FUNCTION_BLOCK FB_Bloque
VAR_INPUT
	Tcheck: TIME := T#1S;
	Treset: TIME := T#1S;
	Tdesplazador: TIME := T#1S;
	Tcinta: TIME := T#0.5S;
END_VAR
VAR_OUTPUT
END_VAR
VAR
	Ciclos: INT;
	Aceptados:INT;
	Rechazados: INT;
	Restantes: INT;
	
	pieza_ok: BOOL;
	
	//Terminal 2
	Pulsador_parada_emergencia AT %I*: BOOL;
	Selector_modo_manual AT %I*: BOOL;
	Pulsador_marcha AT %I*: BOOL;
	Pulsador_parada_NC AT %I*: BOOL;
	Parte_operativa_conectada AT %I*: BOOL;
	Presencia_pale AT %I*: BOOL;
	Codigo_pale_bit_0 AT %I*: BOOL;
	Codigo_pale_bit_1 AT %I*: BOOL;
	
	
	//Terminal 3
	Codigo_pale_bit_2 AT %I*: BOOL;
	Detector_presion AT %I*: BOOL;
	
	//Terminal 4
	Desconecta_parte_operativa AT %Q*: BOOL;
	Lampara_alarma AT %Q*: BOOL;
	Lampara_marcha AT %Q*: BOOL;
	Lampara_falta_material AT %Q*: BOOL;
	Activa_marcha_motor_cinta AT %Q*: BOOL;
	Invierte_marcha_motor_cinta AT %Q*: BOOL;
	Retenedor_pale_baja AT %Q*: BOOL;
	Separador_pale_sube AT %Q*: BOOL;
	
	
	//Terminal 5
 	Avisador_sonoro AT %Q*: BOOL;
	
	//Terminal 6
	Horizontal_descargador_detras AT %I*: BOOL;
	Horizontal_descargador_delante AT %I*: BOOL;
	Vertical_descargador_arriba AT %I*: BOOL;
	Vertical_descargador_abajo AT %I*: BOOL;
	Verificador_arriba AT %I*: BOOL;
	Verificador_abajo AT %I*: BOOL;
	Desplazador_detras AT %I*: BOOL;
	Alimentador_detras AT %I*: BOOL;
	
	
	//Terminal 7
	Alimentador_delante AT %I*: BOOL;
	Vacio_obtenido_vacuostato_descargador AT %I*: BOOL;
	Base_en_Alimentador AT %I*: BOOL;
	
	//Terminal 8
	Descargador_adelante AT %Q*: BOOL;
	Descargador_atras AT %Q*: BOOL;
	Descargador_baja AT %Q*: BOOL;
	Rechazador_adelante AT %Q*: BOOL;
	Verificador_baja AT %Q*: BOOL;
	Desplazador_adelante AT %Q*: BOOL;
	Alimentador_adelante AT %Q*: BOOL;
	Eyector_succiona AT %Q*: BOOL;
	
	NOLAMP: INT;
	t: INT;
	NOTSOUND: INT;
	NOTFOUND: INT;
END_VAR

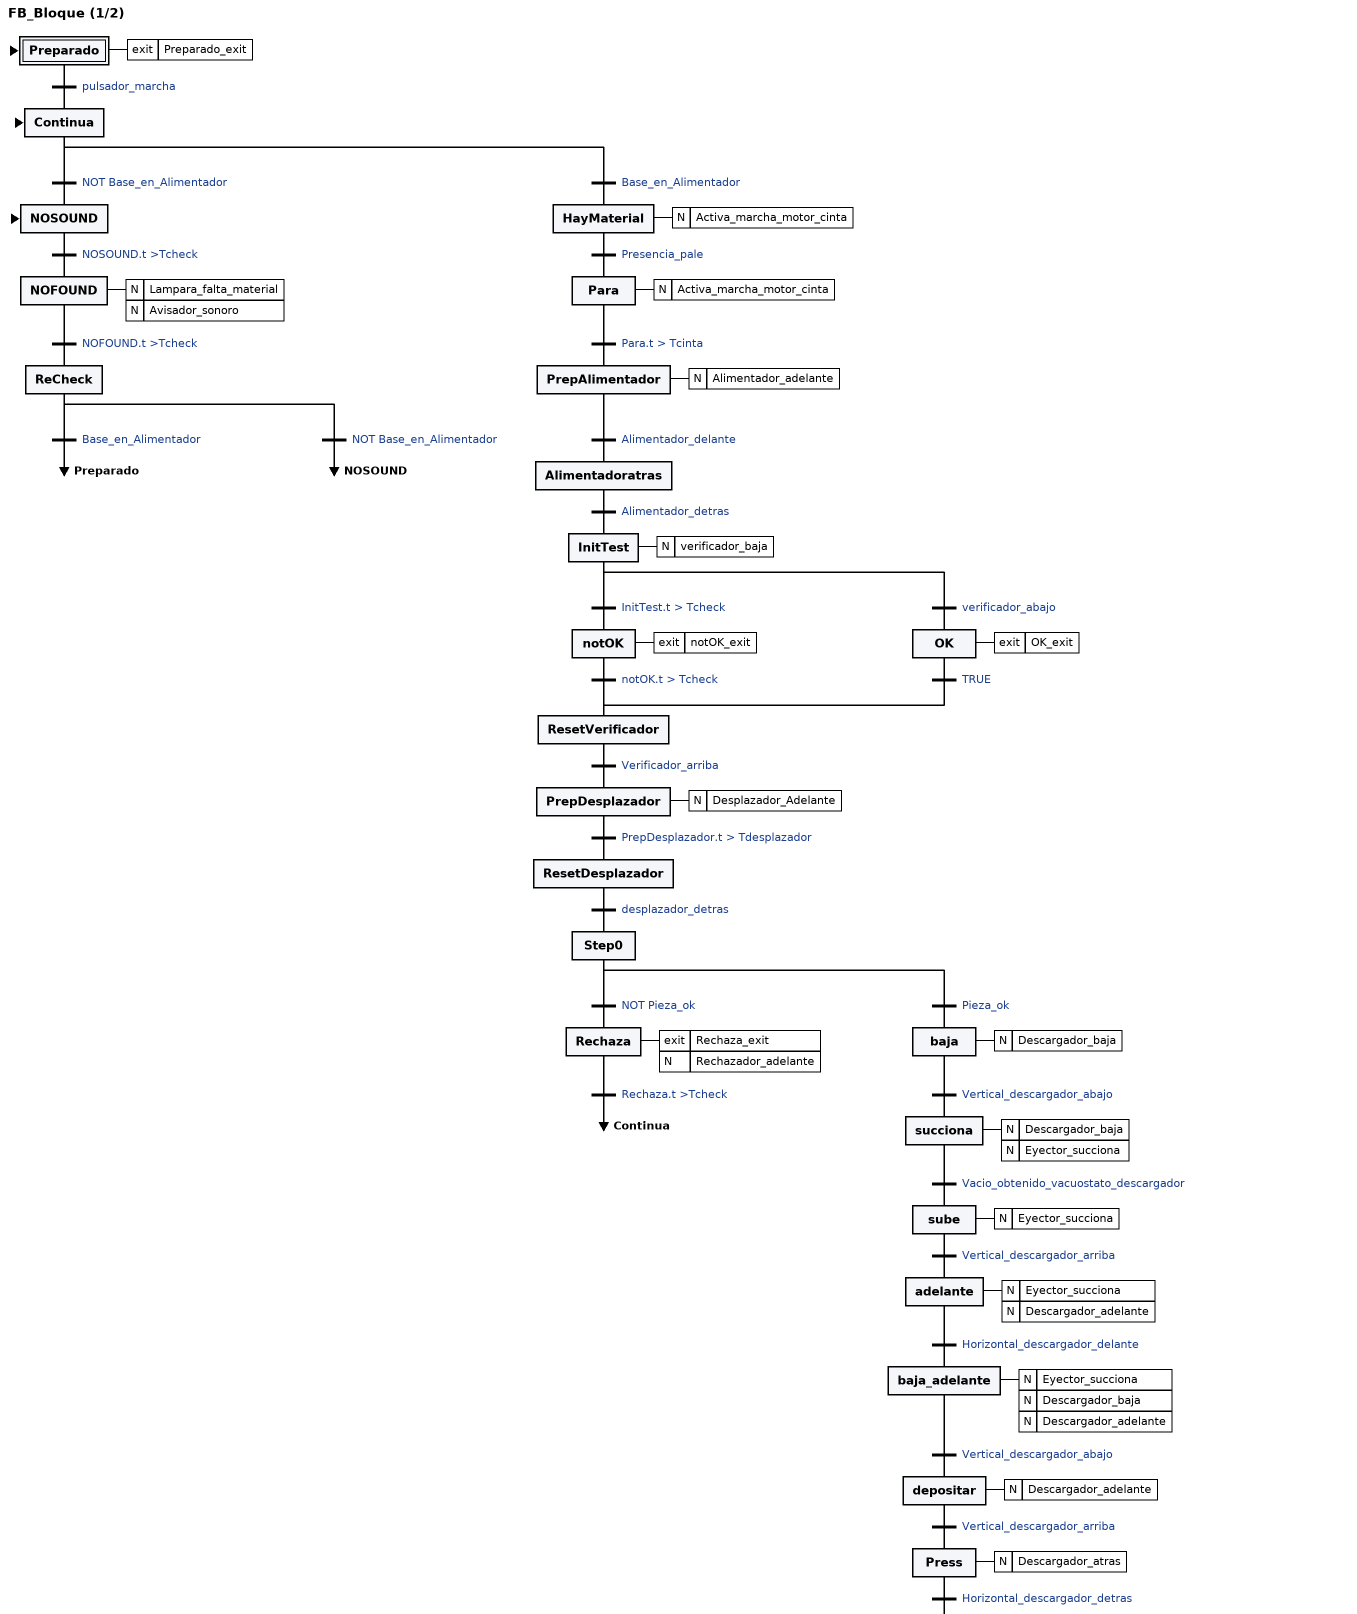
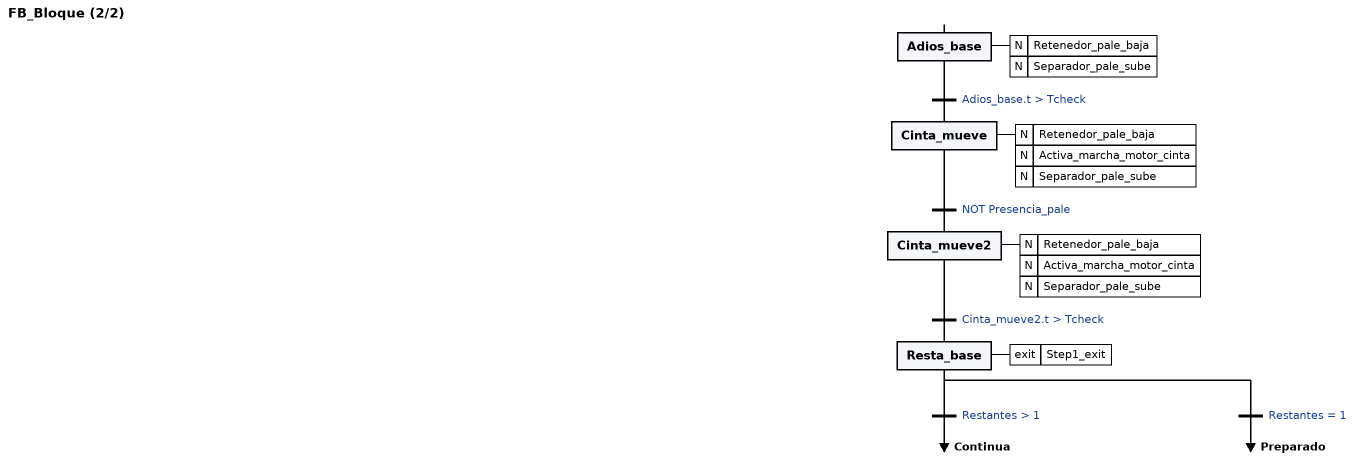
INITIAL_STEP Preparado:
    Preparado_exit(P0);  // exit action
END_STEP
TRANSITION FROM Preparado TO Continua
    := pulsador_marcha;
END_TRANSITION
STEP Continua:
END_STEP
TRANSITION FROM Continua TO NOSOUND
    := NOT Base_en_Alimentador;
END_TRANSITION
STEP NOSOUND:
END_STEP
TRANSITION FROM NOSOUND TO NOFOUND
    := NOSOUND.t >Tcheck;
END_TRANSITION
STEP NOFOUND:
    Lampara_falta_material(N);
    Avisador_sonoro(N);
END_STEP
TRANSITION FROM NOFOUND TO ReCheck
    := NOFOUND.t >Tcheck;
END_TRANSITION
STEP ReCheck:
END_STEP
TRANSITION FROM ReCheck TO Preparado
    := Base_en_Alimentador;
END_TRANSITION
TRANSITION FROM ReCheck TO NOSOUND
    := NOT Base_en_Alimentador;
END_TRANSITION
TRANSITION FROM Continua TO HayMaterial
    := Base_en_Alimentador;
END_TRANSITION
STEP HayMaterial:
    Activa_marcha_motor_cinta(N);
END_STEP
TRANSITION FROM HayMaterial TO Para
    := Presencia_pale;
END_TRANSITION
STEP Para:
    Activa_marcha_motor_cinta(N);
END_STEP
TRANSITION FROM Para TO PrepAlimentador
    := Para.t > Tcinta;
END_TRANSITION
STEP PrepAlimentador:
    Alimentador_adelante(N);
END_STEP
TRANSITION FROM PrepAlimentador TO Alimentadoratras
    := Alimentador_delante;
END_TRANSITION
STEP Alimentadoratras:
END_STEP
TRANSITION FROM Alimentadoratras TO InitTest
    := Alimentador_detras;
END_TRANSITION
STEP InitTest:
    verificador_baja(N);
END_STEP
TRANSITION FROM InitTest TO notOK
    := InitTest.t > Tcheck;
END_TRANSITION
STEP notOK:
    notOK_exit(P0);  // exit action
END_STEP
TRANSITION FROM notOK TO ResetVerificador
    := notOK.t > Tcheck;
END_TRANSITION
TRANSITION FROM InitTest TO OK
    := verificador_abajo;
END_TRANSITION
STEP OK:
    OK_exit(P0);  // exit action
END_STEP
TRANSITION FROM OK TO ResetVerificador
    := TRUE;
END_TRANSITION
STEP ResetVerificador:
END_STEP
TRANSITION FROM ResetVerificador TO PrepDesplazador
    := Verificador_arriba;
END_TRANSITION
STEP PrepDesplazador:
    Desplazador_Adelante(N);
END_STEP
TRANSITION FROM PrepDesplazador TO ResetDesplazador
    := PrepDesplazador.t > Tdesplazador;
END_TRANSITION
STEP ResetDesplazador:
END_STEP
TRANSITION FROM ResetDesplazador TO Step0
    := desplazador_detras;
END_TRANSITION
STEP Step0:
END_STEP
TRANSITION FROM Step0 TO Rechaza
    := NOT Pieza_ok;
END_TRANSITION
STEP Rechaza:
    Rechaza_exit(P0);  // exit action
    Rechazador_adelante(N);
END_STEP
TRANSITION FROM Rechaza TO Continua
    := Rechaza.t >Tcheck;
END_TRANSITION
TRANSITION FROM Step0 TO baja
    := Pieza_ok;
END_TRANSITION
STEP baja:
    Descargador_baja(N);
END_STEP
TRANSITION FROM baja TO succiona
    := Vertical_descargador_abajo;
END_TRANSITION
STEP succiona:
    Descargador_baja(N);
    Eyector_succiona(N);
END_STEP
TRANSITION FROM succiona TO sube
    := Vacio_obtenido_vacuostato_descargador;
END_TRANSITION
STEP sube:
    Eyector_succiona(N);
END_STEP
TRANSITION FROM sube TO adelante
    := Vertical_descargador_arriba;
END_TRANSITION
STEP adelante:
    Eyector_succiona(N);
    Descargador_adelante(N);
END_STEP
TRANSITION FROM adelante TO baja_adelante
    := Horizontal_descargador_delante;
END_TRANSITION
STEP baja_adelante:
    Eyector_succiona(N);
    Descargador_baja(N);
    Descargador_adelante(N);
END_STEP
TRANSITION FROM baja_adelante TO depositar
    := Vertical_descargador_abajo;
END_TRANSITION
STEP depositar:
    Descargador_adelante(N);
END_STEP
TRANSITION FROM depositar TO Press
    := Vertical_descargador_arriba;
END_TRANSITION
STEP Press:
    Descargador_atras(N);
END_STEP
TRANSITION FROM Press TO Adios_base
    := Horizontal_descargador_detras;
END_TRANSITION
STEP Adios_base:
    Retenedor_pale_baja(N);
    Separador_pale_sube(N);
END_STEP
TRANSITION FROM Adios_base TO Cinta_mueve
    := Adios_base.t > Tcheck;
END_TRANSITION
STEP Cinta_mueve:
    Retenedor_pale_baja(N);
    Activa_marcha_motor_cinta(N);
    Separador_pale_sube(N);
END_STEP
TRANSITION FROM Cinta_mueve TO Cinta_mueve2
    := NOT Presencia_pale;
END_TRANSITION
STEP Cinta_mueve2:
    Retenedor_pale_baja(N);
    Activa_marcha_motor_cinta(N);
    Separador_pale_sube(N);
END_STEP
TRANSITION FROM Cinta_mueve2 TO Resta_base
    := Cinta_mueve2.t > Tcheck;
END_TRANSITION
STEP Resta_base:
    Step1_exit(P0);  // exit action
END_STEP
TRANSITION FROM Resta_base TO Continua
    := Restantes > 1;
END_TRANSITION
TRANSITION FROM Resta_base TO Preparado
    := Restantes = 1;
END_TRANSITION

ACTION notOK_exit:
pieza_ok := FALSE;
END_ACTION

ACTION OK_exit:
pieza_ok := true;
END_ACTION

ACTION Preparado_entry:
//Ciclos:= 3;
Rechazados :=0;
Aceptados :=0;
Restantes:=Ciclos;
END_ACTION

ACTION Preparado_exit:
IF Restantes = 0 THEN

	Restantes := Ciclos;
	Aceptados := 0;
	Rechazados := 0;	

END_IF
END_ACTION

ACTION Rechaza_exit:
Rechazados:= Rechazados+1;
END_ACTION

ACTION Step1_exit:
Aceptados:=Aceptados+1;
Restantes:=Restantes-1;
END_ACTION

END_FUNCTION_BLOCK

(* stored: Version 1.1.0.1, ProductVersion 3.1.4024.12
   POU FB_Bloque: Id {ec5bfe8f-5238-4cef-82c6-2f925b841434}, SpecialFunc None
   Action notOK_exit: Id {07375664-efc3-4adf-b0b0-a037ed282644}
   Action OK_exit: Id {71fdc0d3-9a4d-43a1-9501-ea0ef3b2e92a}
   Action Preparado_entry: Id {c24d1924-ac38-41b9-809d-9a84317adff6}
   Action Preparado_exit: Id {a52776b1-983b-4aa6-a045-4f3bfb6c1896}
   Action Rechaza_exit: Id {f753a87a-6ed7-4fd8-92ae-0c27075b215f}
   Action Step1_exit: Id {7ab2790f-e6a7-4cf7-a12c-3fff6a637426} *)
